PROGRAM MAIN
VAR
	ManualControl_0: ManualControl;
	AutomaticControl_0: AutomaticControl;
END_VAR

// Initially it goes to position (0,0,0,0) and initializes motors by Initialize PRG.
// There is Safety PRG that keeps checking if motors are out of bounds.
// Motors are instantiated as global vars to retain their properties.
// CountCurrentPosition PRG is the only place where we count position using the sensors.
// RestorePreviousAutomaticState is a FB that gets execture cyclic until all the directions are set to previous positions.
// AutomaticControl FB remembers which recipe is being executed and recipe remembers its state.
VAR // added by the converter: edge detectors and wires of the graphical bodies
    _ft1 : F_TRIG;
    _rt1 : R_TRIG;
    _w1 : BOOL;
END_VAR

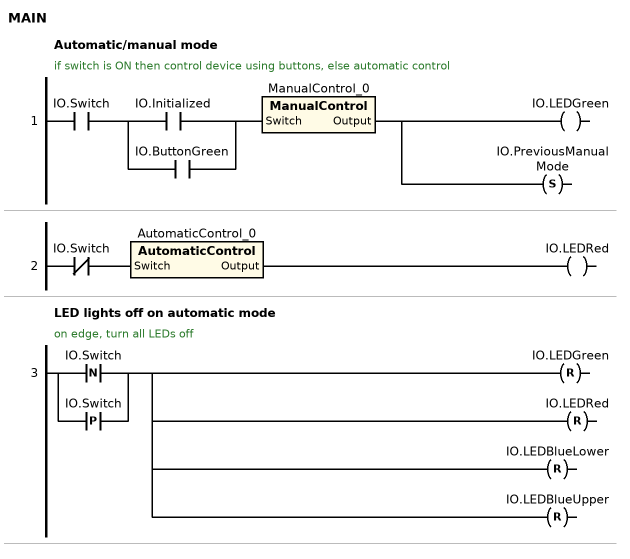
// NETWORK 1: Automatic/manual mode
// if switch is ON then control device using buttons, else automatic control
ManualControl_0(Switch := IO.Switch AND IO.Initialized OR IO.Switch AND IO.ButtonGreen); // ManualControl
IO.LEDGreen := ManualControl_0.Output;
IO.PreviousManualMode S= ManualControl_0.Output;

// NETWORK 2
AutomaticControl_0(Switch := NOT IO.Switch); // AutomaticControl
IO.LEDRed := AutomaticControl_0.Output;

// NETWORK 3: LED lights off on automatic mode
// on edge, turn all LEDs off
_ft1(CLK := IO.Switch);
_rt1(CLK := IO.Switch);
_w1 := _ft1.Q OR _rt1.Q;
IO.LEDGreen R= _w1;
IO.LEDRed R= _w1;
IO.LEDBlueLower R= _w1;
IO.LEDBlueUpper R= _w1;

END_PROGRAM

(* stored: Version 1.1.0.1, ProductVersion 3.1.4024.13
   POU MAIN: Id {ca0d1193-1c86-427a-9c71-41bf6bccd822}, SpecialFunc None *)
